(* Logix 5000 project; controller cal1632 1756-L62 rev 16.20; software revision 16.05; part 10 of 57 *)
(* tags used below, declared in another part *)
   FAULT : BOOL;
   HMI : BOOL;
   p01_sys_scp : SYS_SCP;
   p01r02 : routine;
   p01r09_pb_global_reset : BOOL;
   p11_ai_exh_amps : REAL;
   p11_ai_exh_hz : REAL;
   p11_ai_exh_hz_max : REAL;
   p11_ai_exh_rpm : REAL;
   p11_ai_lfl : REAL;
   p11_ai_prs : REAL;
   p11_ai_recirc_amps : REAL;
   p11_ai_recirc_hz : REAL;
   p11_ai_recirc_hz_max : REAL;
   p11_ai_recirc_rpm : REAL;
   p11_ai_tc01 : REAL;
   p11_ai_tc02 : REAL;
   p11_ao_cv : REAL;
   p11_ao_exhaust_selected_speed : REAL;
   p11_ao_recirc_selected_speed : REAL;
   p11_di_burner_auto : BOOL;
   p11_di_burner_safeties_ok : BOOL;
   p11_di_door_open : BOOL;
   p11_di_exh : acs800_di_normal;
   p11_di_exh_fan_mtr_ts : BOOL;
   p11_di_exh_flow_ok : BOOL;
   p11_di_flame_failure : BOOL;
   p11_di_flame_on : BOOL;
   p11_di_fresh_air_clean : BOOL;
   p11_di_high_limit_temp_ok : BOOL;
   p11_di_recirc : acs800_di_normal;
   p11_di_recirc_fan_mtr_ts : BOOL;
   p11_di_recirc_flow_ok : BOOL;
   p11_di_sp0 : BOOL;
   p11_di_sp00 : BOOL;
   p11_di_sp1 : BOOL;
   p11_di_sp2 : BOOL;
   p11_di_sp3 : BOOL;
   p11_di_tc01_bo : BOOL;
   p11_di_tc02_bo : BOOL;
   p11_di_zone_air_clean : BOOL;
   p11_dint_to_hmi : DINT[16];
   p11_do_enable_burner : BOOL;
   p11_do_exh : acs800_do_normal;
   p11_do_recirc : acs800_do_normal;
   p11_do_rst_flame : BOOL;
   p11_exhaust_input_max : REAL;
   p11_exhaust_input_min : REAL;
   p11_exhaust_output_max : REAL;
   p11_exhaust_output_min : REAL;
   p11_hc_input_max : REAL;
   p11_hc_input_min : REAL;
   p11_hc_output_max : REAL;
   p11_hc_output_min : REAL;
   p11_lfl_input_max : REAL;
   p11_lfl_input_min : REAL;
   p11_lfl_output_max : REAL;
   p11_lfl_output_min : REAL;
   p11_param_tc01z : REAL;
   p11_param_tc02z : REAL;
   p11_prs_input_max : REAL;
   p11_prs_input_min : REAL;
   p11_prs_output_max : REAL;
   p11_prs_output_min : REAL;
   p11_recirc_input_max : REAL;
   p11_recirc_input_min : REAL;
   p11_recirc_output_max : REAL;
   p11_recirc_output_min : REAL;
   p11r03 : routine;
   p11r03_hz : SYS_SCP;
   p11r03_timer_fault : TIMER[4];
   p11r03_timer_warning : TIMER[4];
   p11r04 : routine;
   p11r04_timer_fault : TIMER[4];
   p11r04_timer_warning : TIMER[4];
   p11r05 : routine;
   p11r05_exh_status : DINT;
   p11r05_recirc_status : DINT;
   p11r05_temp_ctrl_status : DINT;
   p11r05_timer_fault : TIMER[4];
   p11r05_timer_warning : TIMER[4];
   p11r20_state : DINT;
   p11r20_status : DINT;
   p11r30 : routine;
   p11r30_permissive_run : BOOL;
   p11r30_request_heat : BOOL;
   p11r30_request_manual : BOOL;
   p11r30_vfds_ready : BOOL;
   p11r31 : routine;
   p11r31_request_auto_run : BOOL;
   p11r31_request_auto_stop : BOOL;
   p11r31_vfd_stopped : BOOL;
   p11r32 : routine;
   p11r32_request_auto_run : BOOL;
   p11r32_request_auto_stop : BOOL;
   p11r32_vfd_stopped : BOOL;
(* P11_Zone_1, continued *)

ROUTINE R03_Input   (* ladder *)
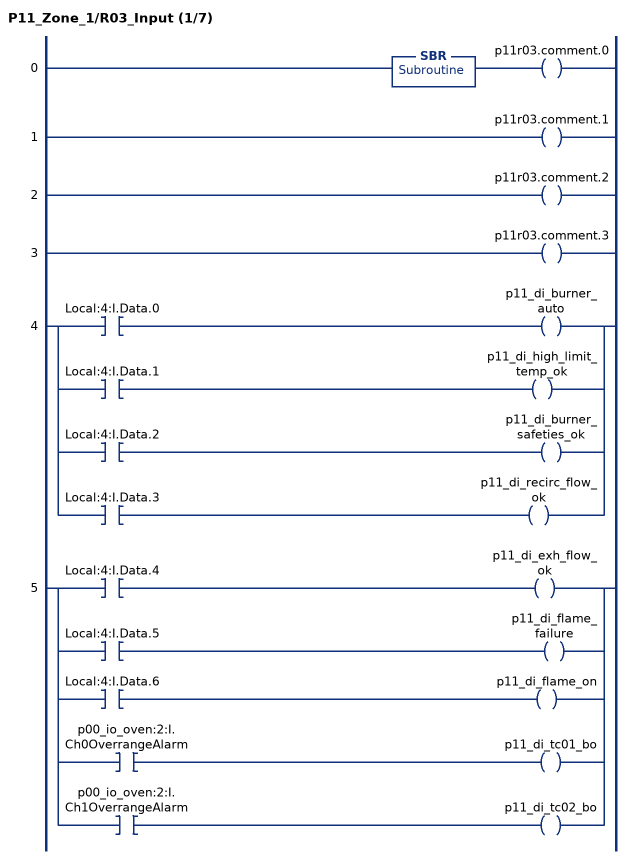
   0: SBR()OTE(p11r03.comment.0);
   1: OTE(p11r03.comment.1);
   2: OTE(p11r03.comment.2);
   3: OTE(p11r03.comment.3);
   4: [XIC(Local:4:I.Data.0) OTE(p11_di_burner_auto) ,XIC(Local:4:I.Data.1) OTE(p11_di_high_limit_temp_ok) ,XIC(Local:4:I.Data.2) OTE(p11_di_burner_safeties_ok) ,XIC(Local:4:I.Data.3) OTE(p11_di_recirc_flow_ok) ];
   5: [XIC(Local:4:I.Data.4) OTE(p11_di_exh_flow_ok) ,XIC(Local:4:I.Data.5) OTE(p11_di_flame_failure) ,XIC(Local:4:I.Data.6) OTE(p11_di_flame_on) ,XIC(p00_io_oven:2:I.Ch0OverrangeAlarm) OTE(p11_di_tc01_bo) ,XIC(p00_io_oven:2:I.Ch1OverrangeAlarm) OTE(p11_di_tc02_bo) ];
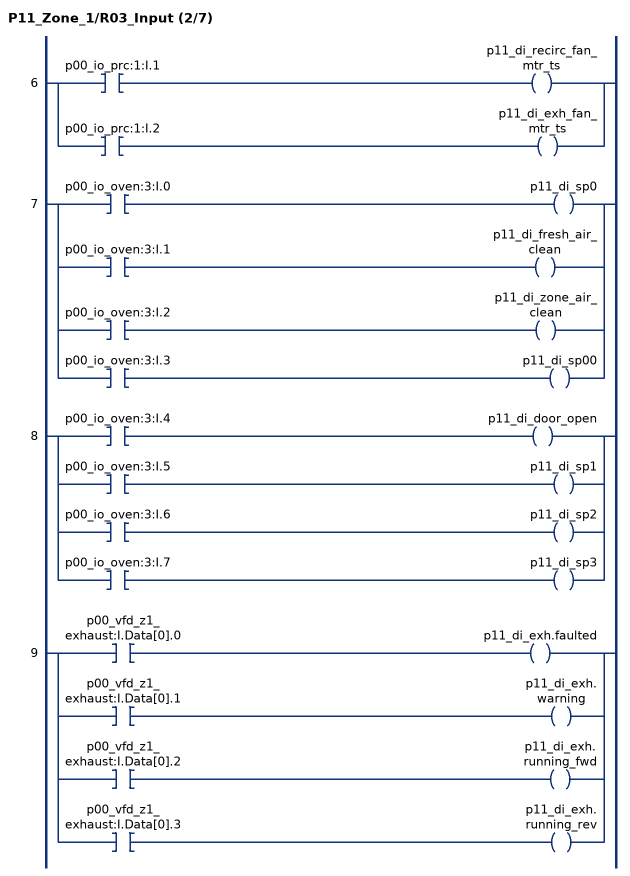
   6: [XIC(p00_io_prc:1:I.1) OTE(p11_di_recirc_fan_mtr_ts) ,XIC(p00_io_prc:1:I.2) OTE(p11_di_exh_fan_mtr_ts) ];
   7: [XIC(p00_io_oven:3:I.0) OTE(p11_di_sp0) ,XIC(p00_io_oven:3:I.1) OTE(p11_di_fresh_air_clean) ,XIC(p00_io_oven:3:I.2) OTE(p11_di_zone_air_clean) ,XIC(p00_io_oven:3:I.3) OTE(p11_di_sp00) ];
   8: [XIC(p00_io_oven:3:I.4) OTE(p11_di_door_open) ,XIC(p00_io_oven:3:I.5) OTE(p11_di_sp1) ,XIC(p00_io_oven:3:I.6) OTE(p11_di_sp2) ,XIC(p00_io_oven:3:I.7) OTE(p11_di_sp3) ];
   9: [XIC(p00_vfd_z1_exhaust:I.Data[0].0) OTE(p11_di_exh.faulted) ,XIC(p00_vfd_z1_exhaust:I.Data[0].1) OTE(p11_di_exh.warning) ,XIC(p00_vfd_z1_exhaust:I.Data[0].2) OTE(p11_di_exh.running_fwd) ,XIC(p00_vfd_z1_exhaust:I.Data[0].3) OTE(p11_di_exh.running_rev) ];
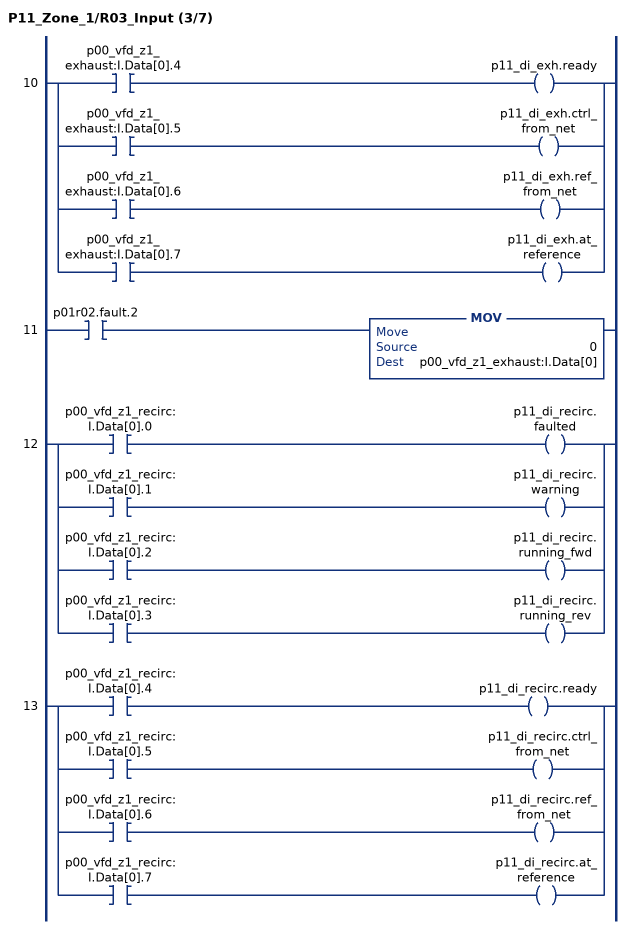
   10: [XIC(p00_vfd_z1_exhaust:I.Data[0].4) OTE(p11_di_exh.ready) ,XIC(p00_vfd_z1_exhaust:I.Data[0].5) OTE(p11_di_exh.ctrl_from_net) ,XIC(p00_vfd_z1_exhaust:I.Data[0].6) OTE(p11_di_exh.ref_from_net) ,XIC(p00_vfd_z1_exhaust:I.Data[0].7) OTE(p11_di_exh.at_reference) ];
   11: XIC(p01r02.fault.2)MOV(0,p00_vfd_z1_exhaust:I.Data[0]);
   12: [XIC(p00_vfd_z1_recirc:I.Data[0].0) OTE(p11_di_recirc.faulted) ,XIC(p00_vfd_z1_recirc:I.Data[0].1) OTE(p11_di_recirc.warning) ,XIC(p00_vfd_z1_recirc:I.Data[0].2) OTE(p11_di_recirc.running_fwd) ,XIC(p00_vfd_z1_recirc:I.Data[0].3) OTE(p11_di_recirc.running_rev) ];
   13: [XIC(p00_vfd_z1_recirc:I.Data[0].4) OTE(p11_di_recirc.ready) ,XIC(p00_vfd_z1_recirc:I.Data[0].5) OTE(p11_di_recirc.ctrl_from_net) ,XIC(p00_vfd_z1_recirc:I.Data[0].6) OTE(p11_di_recirc.ref_from_net) ,XIC(p00_vfd_z1_recirc:I.Data[0].7) OTE(p11_di_recirc.at_reference) ];
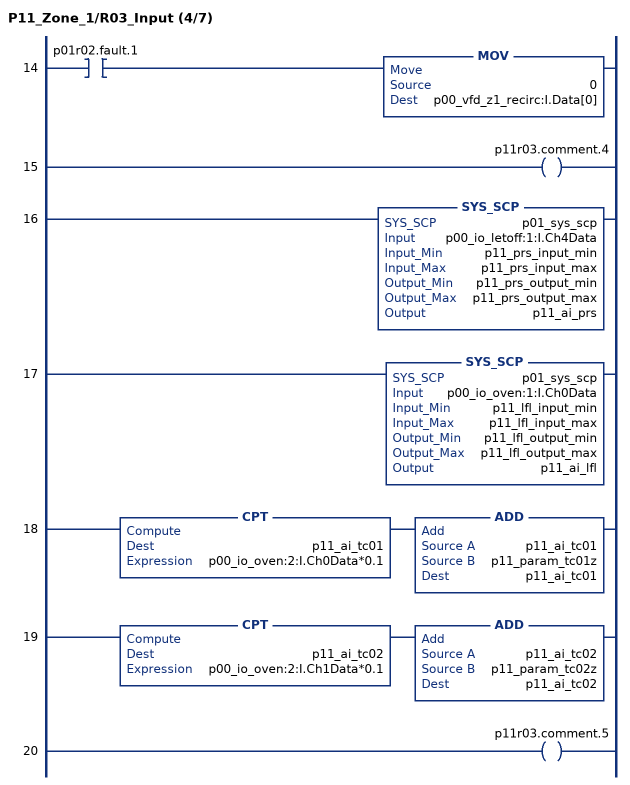
   14: XIC(p01r02.fault.1)MOV(0,p00_vfd_z1_recirc:I.Data[0]);
   15: OTE(p11r03.comment.4);
   16: SYS_SCP(p01_sys_scp,p00_io_letoff:1:I.Ch4Data,p11_prs_input_min,p11_prs_input_max,p11_prs_output_min,p11_prs_output_max,p11_ai_prs);
   17: SYS_SCP(p01_sys_scp,p00_io_oven:1:I.Ch0Data,p11_lfl_input_min,p11_lfl_input_max,p11_lfl_output_min,p11_lfl_output_max,p11_ai_lfl);
   18: CPT(p11_ai_tc01,p00_io_oven:2:I.Ch0Data*0.1)ADD(p11_ai_tc01,p11_param_tc01z,p11_ai_tc01);
   19: CPT(p11_ai_tc02,p00_io_oven:2:I.Ch1Data*0.1)ADD(p11_ai_tc02,p11_param_tc02z,p11_ai_tc02);
   20: OTE(p11r03.comment.5);
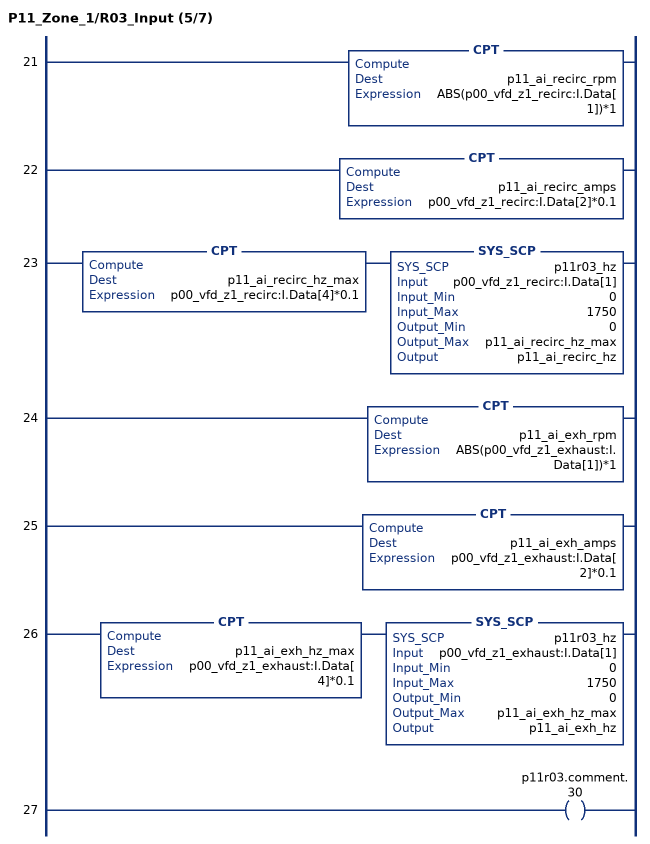
   21: CPT(p11_ai_recirc_rpm,ABS(p00_vfd_z1_recirc:I.Data[1])*1);
   22: CPT(p11_ai_recirc_amps,p00_vfd_z1_recirc:I.Data[2]*0.1);
   23: CPT(p11_ai_recirc_hz_max,p00_vfd_z1_recirc:I.Data[4]*0.1)SYS_SCP(p11r03_hz,p00_vfd_z1_recirc:I.Data[1],0,1750,0,p11_ai_recirc_hz_max,p11_ai_recirc_hz);
   24: CPT(p11_ai_exh_rpm,ABS(p00_vfd_z1_exhaust:I.Data[1])*1);
   25: CPT(p11_ai_exh_amps,p00_vfd_z1_exhaust:I.Data[2]*0.1);
   26: CPT(p11_ai_exh_hz_max,p00_vfd_z1_exhaust:I.Data[4]*0.1)SYS_SCP(p11r03_hz,p00_vfd_z1_exhaust:I.Data[1],0,1750,0,p11_ai_exh_hz_max,p11_ai_exh_hz);
   27: OTE(p11r03.comment.30);
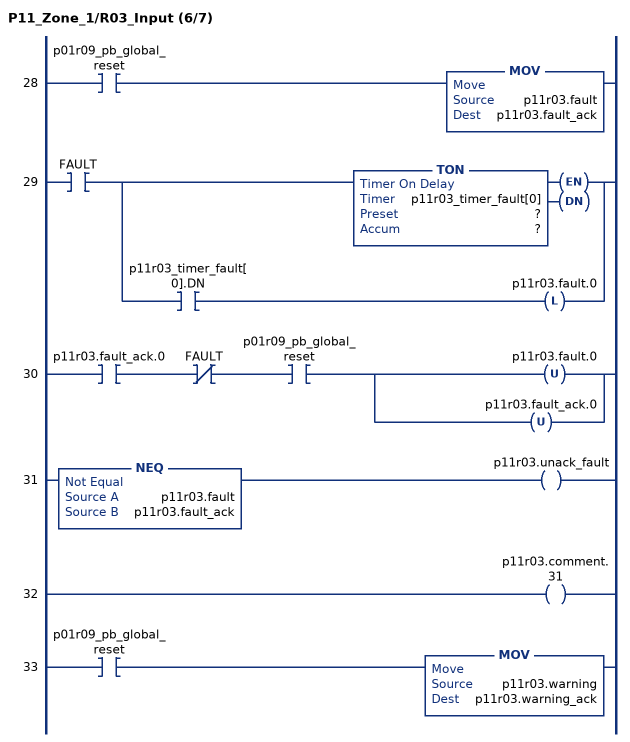
   28: XIC(p01r09_pb_global_reset)MOV(p11r03.fault,p11r03.fault_ack);
   29: XIC(FAULT)[TON(p11r03_timer_fault[0],?,?) ,XIC(p11r03_timer_fault[0].DN) OTL(p11r03.fault.0) ];
   30: XIC(p11r03.fault_ack.0)XIO(FAULT)XIC(p01r09_pb_global_reset)[OTU(p11r03.fault.0) ,OTU(p11r03.fault_ack.0) ];
   31: NEQ(p11r03.fault,p11r03.fault_ack)OTE(p11r03.unack_fault);
   32: OTE(p11r03.comment.31);
   33: XIC(p01r09_pb_global_reset)MOV(p11r03.warning,p11r03.warning_ack);
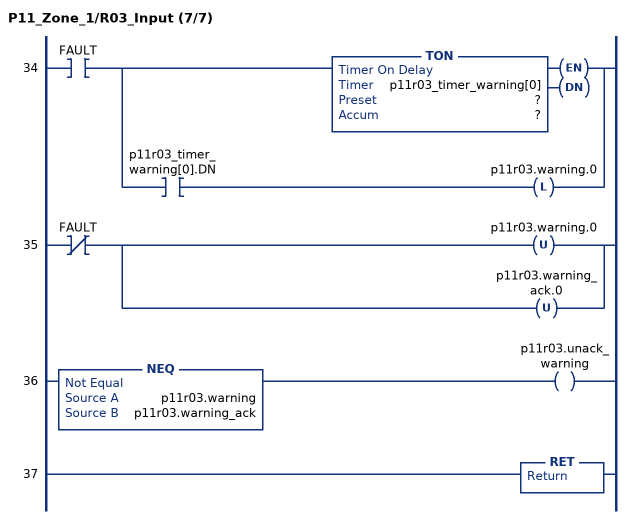
   34: XIC(FAULT)[TON(p11r03_timer_warning[0],?,?) ,XIC(p11r03_timer_warning[0].DN) OTL(p11r03.warning.0) ];
   35: XIO(FAULT)[OTU(p11r03.warning.0) ,OTU(p11r03.warning_ack.0) ];
   36: NEQ(p11r03.warning,p11r03.warning_ack)OTE(p11r03.unack_warning);
   37: RET();
END_ROUTINE

ROUTINE R04_Output   (* ladder *)
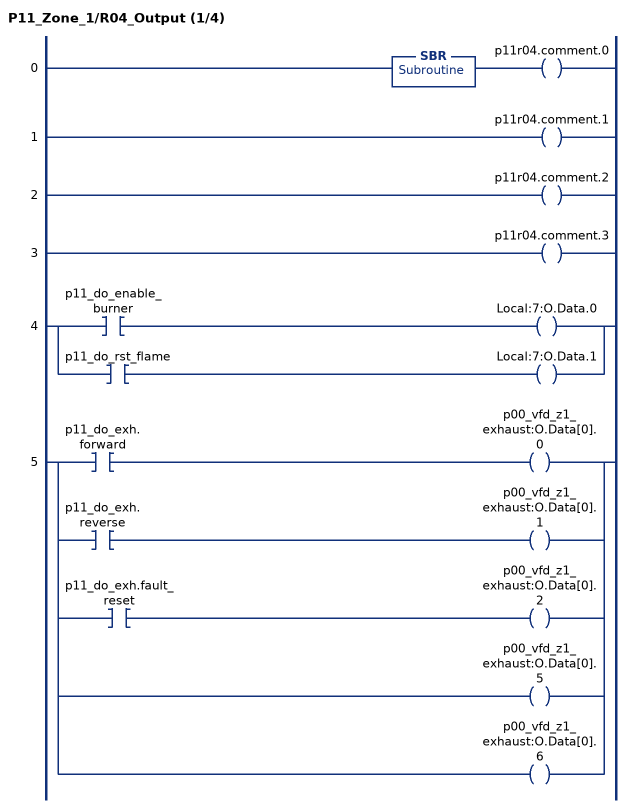
   0: SBR()OTE(p11r04.comment.0);
   1: OTE(p11r04.comment.1);
   2: OTE(p11r04.comment.2);
   3: OTE(p11r04.comment.3);
   4: [XIC(p11_do_enable_burner) OTE(Local:7:O.Data.0) ,XIC(p11_do_rst_flame) OTE(Local:7:O.Data.1) ];
   5: [XIC(p11_do_exh.forward) OTE(p00_vfd_z1_exhaust:O.Data[0].0) ,XIC(p11_do_exh.reverse) OTE(p00_vfd_z1_exhaust:O.Data[0].1) ,XIC(p11_do_exh.fault_reset) OTE(p00_vfd_z1_exhaust:O.Data[0].2) ,OTE(p00_vfd_z1_exhaust:O.Data[0].5) ,OTE(p00_vfd_z1_exhaust:O.Data[0].6) ];
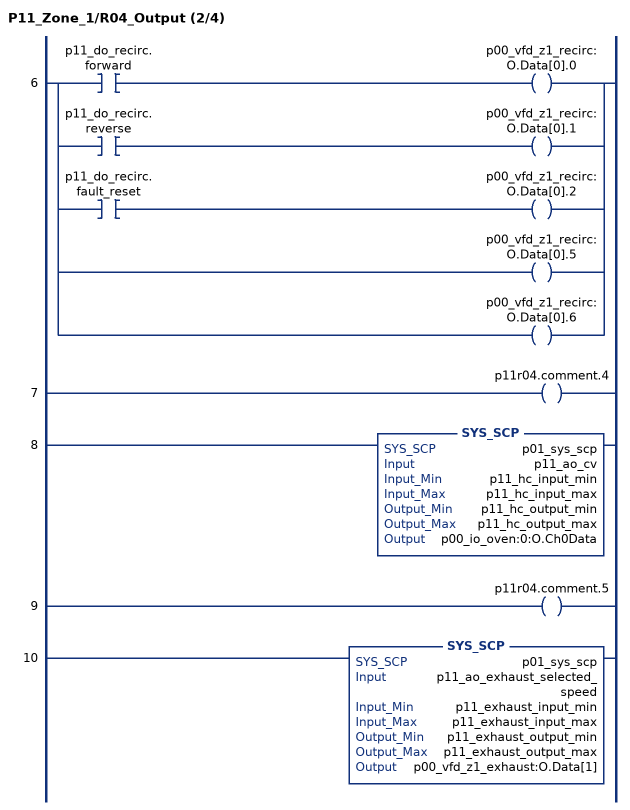
   6: [XIC(p11_do_recirc.forward) OTE(p00_vfd_z1_recirc:O.Data[0].0) ,XIC(p11_do_recirc.reverse) OTE(p00_vfd_z1_recirc:O.Data[0].1) ,XIC(p11_do_recirc.fault_reset) OTE(p00_vfd_z1_recirc:O.Data[0].2) ,OTE(p00_vfd_z1_recirc:O.Data[0].5) ,OTE(p00_vfd_z1_recirc:O.Data[0].6) ];
   7: OTE(p11r04.comment.4);
   8: SYS_SCP(p01_sys_scp,p11_ao_cv,p11_hc_input_min,p11_hc_input_max,p11_hc_output_min,p11_hc_output_max,p00_io_oven:0:O.Ch0Data);
   9: OTE(p11r04.comment.5);
   10: SYS_SCP(p01_sys_scp,p11_ao_exhaust_selected_speed,p11_exhaust_input_min,p11_exhaust_input_max,p11_exhaust_output_min,p11_exhaust_output_max,p00_vfd_z1_exhaust:O.Data[1]);
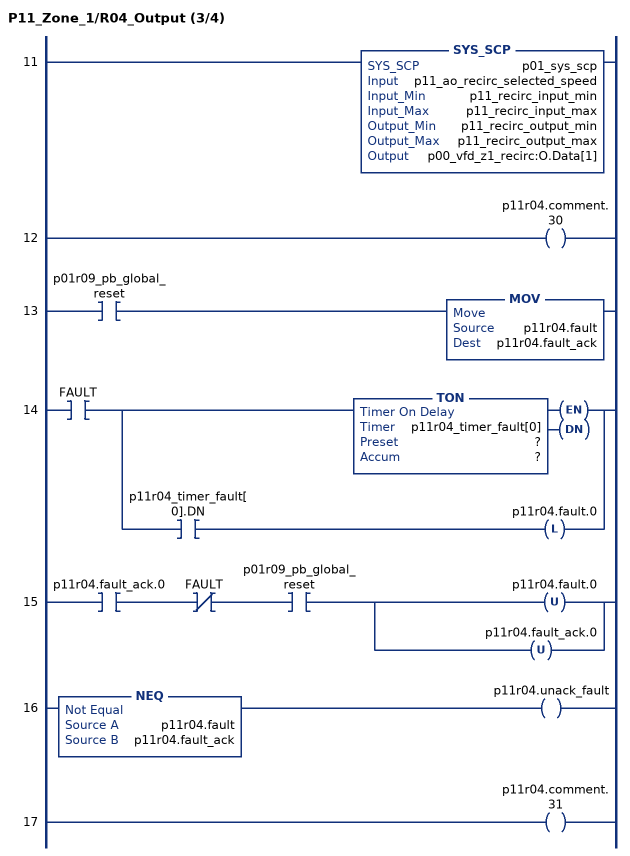
   11: SYS_SCP(p01_sys_scp,p11_ao_recirc_selected_speed,p11_recirc_input_min,p11_recirc_input_max,p11_recirc_output_min,p11_recirc_output_max,p00_vfd_z1_recirc:O.Data[1]);
   12: OTE(p11r04.comment.30);
   13: XIC(p01r09_pb_global_reset)MOV(p11r04.fault,p11r04.fault_ack);
   14: XIC(FAULT)[TON(p11r04_timer_fault[0],?,?) ,XIC(p11r04_timer_fault[0].DN) OTL(p11r04.fault.0) ];
   15: XIC(p11r04.fault_ack.0)XIO(FAULT)XIC(p01r09_pb_global_reset)[OTU(p11r04.fault.0) ,OTU(p11r04.fault_ack.0) ];
   16: NEQ(p11r04.fault,p11r04.fault_ack)OTE(p11r04.unack_fault);
   17: OTE(p11r04.comment.31);
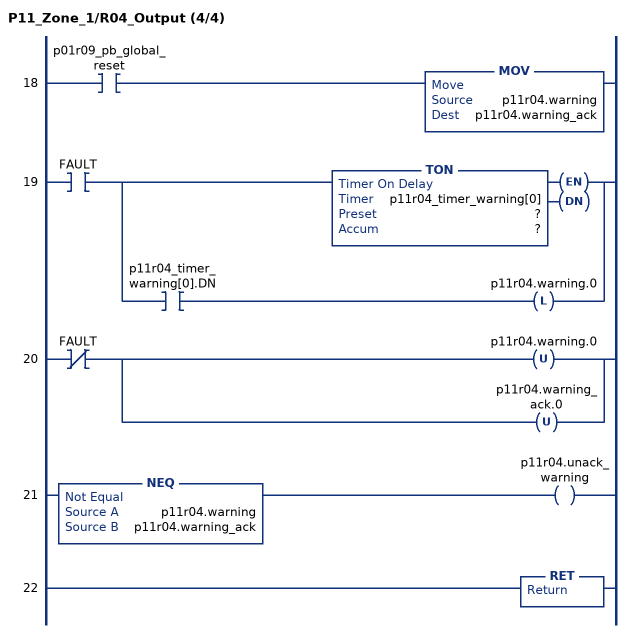
   18: XIC(p01r09_pb_global_reset)MOV(p11r04.warning,p11r04.warning_ack);
   19: XIC(FAULT)[TON(p11r04_timer_warning[0],?,?) ,XIC(p11r04_timer_warning[0].DN) OTL(p11r04.warning.0) ];
   20: XIO(FAULT)[OTU(p11r04.warning.0) ,OTU(p11r04.warning_ack.0) ];
   21: NEQ(p11r04.warning,p11r04.warning_ack)OTE(p11r04.unack_warning);
   22: RET();
END_ROUTINE

ROUTINE R05_Dint_to_HMI   (* ladder *)
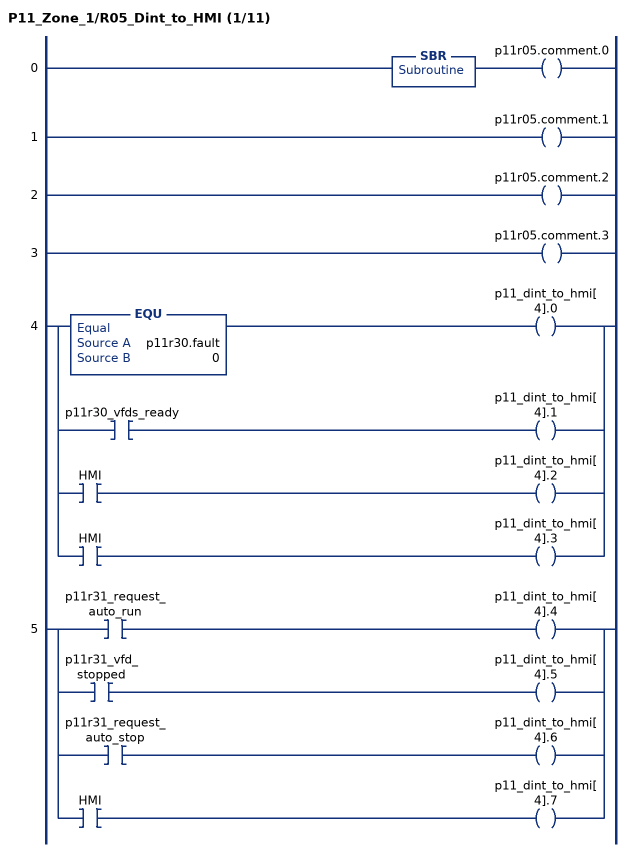
   0: SBR()OTE(p11r05.comment.0);
   1: OTE(p11r05.comment.1);
   2: OTE(p11r05.comment.2);
   3: OTE(p11r05.comment.3);
   4: [EQU(p11r30.fault,0) OTE(p11_dint_to_hmi[4].0) ,XIC(p11r30_vfds_ready) OTE(p11_dint_to_hmi[4].1) ,XIC(HMI) OTE(p11_dint_to_hmi[4].2) ,XIC(HMI) OTE(p11_dint_to_hmi[4].3) ];
   5: [XIC(p11r31_request_auto_run) OTE(p11_dint_to_hmi[4].4) ,XIC(p11r31_vfd_stopped) OTE(p11_dint_to_hmi[4].5) ,XIC(p11r31_request_auto_stop) OTE(p11_dint_to_hmi[4].6) ,XIC(HMI) OTE(p11_dint_to_hmi[4].7) ];
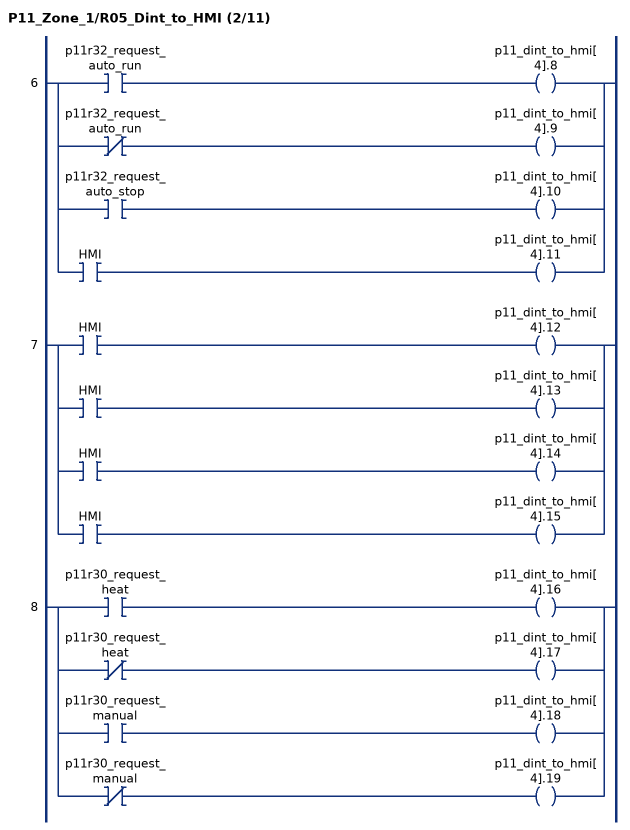
   6: [XIC(p11r32_request_auto_run) OTE(p11_dint_to_hmi[4].8) ,XIO(p11r32_request_auto_run) OTE(p11_dint_to_hmi[4].9) ,XIC(p11r32_request_auto_stop) OTE(p11_dint_to_hmi[4].10) ,XIC(HMI) OTE(p11_dint_to_hmi[4].11) ];
   7: [XIC(HMI) OTE(p11_dint_to_hmi[4].12) ,XIC(HMI) OTE(p11_dint_to_hmi[4].13) ,XIC(HMI) OTE(p11_dint_to_hmi[4].14) ,XIC(HMI) OTE(p11_dint_to_hmi[4].15) ];
   8: [XIC(p11r30_request_heat) OTE(p11_dint_to_hmi[4].16) ,XIO(p11r30_request_heat) OTE(p11_dint_to_hmi[4].17) ,XIC(p11r30_request_manual) OTE(p11_dint_to_hmi[4].18) ,XIO(p11r30_request_manual) OTE(p11_dint_to_hmi[4].19) ];
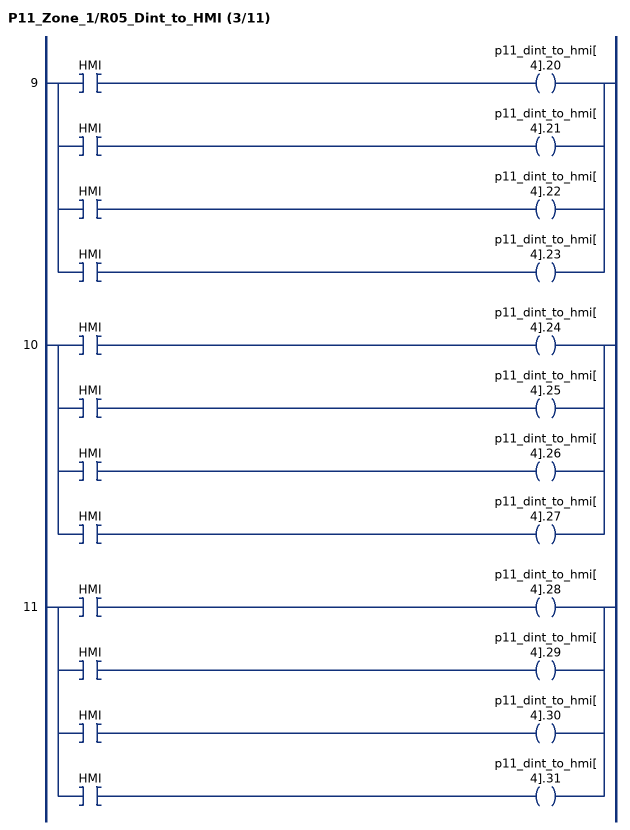
   9: [XIC(HMI) OTE(p11_dint_to_hmi[4].20) ,XIC(HMI) OTE(p11_dint_to_hmi[4].21) ,XIC(HMI) OTE(p11_dint_to_hmi[4].22) ,XIC(HMI) OTE(p11_dint_to_hmi[4].23) ];
   10: [XIC(HMI) OTE(p11_dint_to_hmi[4].24) ,XIC(HMI) OTE(p11_dint_to_hmi[4].25) ,XIC(HMI) OTE(p11_dint_to_hmi[4].26) ,XIC(HMI) OTE(p11_dint_to_hmi[4].27) ];
   11: [XIC(HMI) OTE(p11_dint_to_hmi[4].28) ,XIC(HMI) OTE(p11_dint_to_hmi[4].29) ,XIC(HMI) OTE(p11_dint_to_hmi[4].30) ,XIC(HMI) OTE(p11_dint_to_hmi[4].31) ];
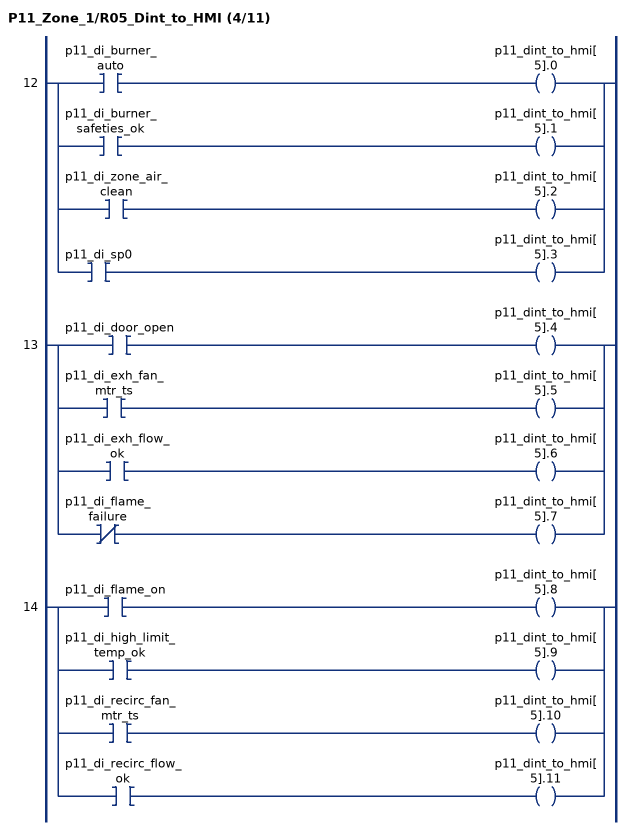
   12: [XIC(p11_di_burner_auto) OTE(p11_dint_to_hmi[5].0) ,XIC(p11_di_burner_safeties_ok) OTE(p11_dint_to_hmi[5].1) ,XIC(p11_di_zone_air_clean) OTE(p11_dint_to_hmi[5].2) ,XIC(p11_di_sp0) OTE(p11_dint_to_hmi[5].3) ];
   13: [XIC(p11_di_door_open) OTE(p11_dint_to_hmi[5].4) ,XIC(p11_di_exh_fan_mtr_ts) OTE(p11_dint_to_hmi[5].5) ,XIC(p11_di_exh_flow_ok) OTE(p11_dint_to_hmi[5].6) ,XIO(p11_di_flame_failure) OTE(p11_dint_to_hmi[5].7) ];
   14: [XIC(p11_di_flame_on) OTE(p11_dint_to_hmi[5].8) ,XIC(p11_di_high_limit_temp_ok) OTE(p11_dint_to_hmi[5].9) ,XIC(p11_di_recirc_fan_mtr_ts) OTE(p11_dint_to_hmi[5].10) ,XIC(p11_di_recirc_flow_ok) OTE(p11_dint_to_hmi[5].11) ];
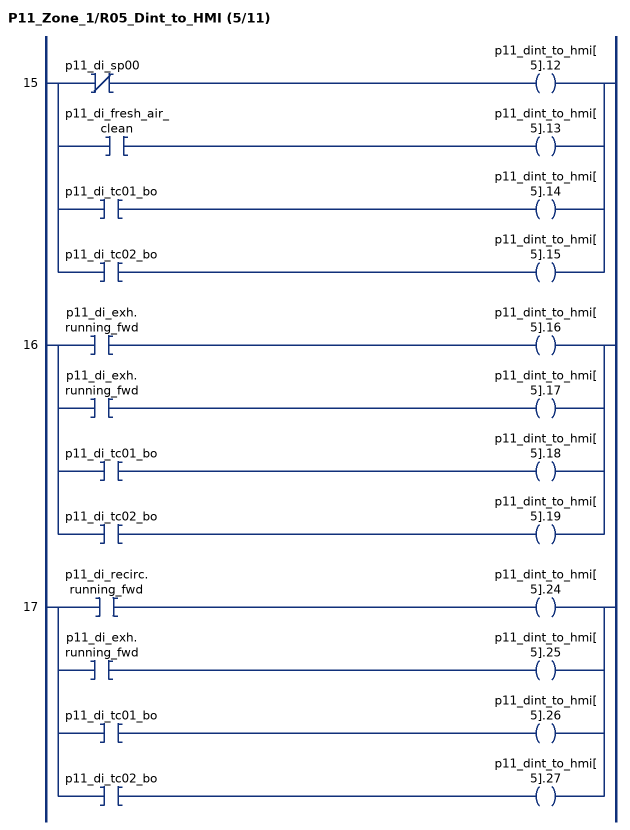
   15: [XIO(p11_di_sp00) OTE(p11_dint_to_hmi[5].12) ,XIC(p11_di_fresh_air_clean) OTE(p11_dint_to_hmi[5].13) ,XIC(p11_di_tc01_bo) OTE(p11_dint_to_hmi[5].14) ,XIC(p11_di_tc02_bo) OTE(p11_dint_to_hmi[5].15) ];
   16: [XIC(p11_di_exh.running_fwd) OTE(p11_dint_to_hmi[5].16) ,XIC(p11_di_exh.running_fwd) OTE(p11_dint_to_hmi[5].17) ,XIC(p11_di_tc01_bo) OTE(p11_dint_to_hmi[5].18) ,XIC(p11_di_tc02_bo) OTE(p11_dint_to_hmi[5].19) ];
   17: [XIC(p11_di_recirc.running_fwd) OTE(p11_dint_to_hmi[5].24) ,XIC(p11_di_exh.running_fwd) OTE(p11_dint_to_hmi[5].25) ,XIC(p11_di_tc01_bo) OTE(p11_dint_to_hmi[5].26) ,XIC(p11_di_tc02_bo) OTE(p11_dint_to_hmi[5].27) ];
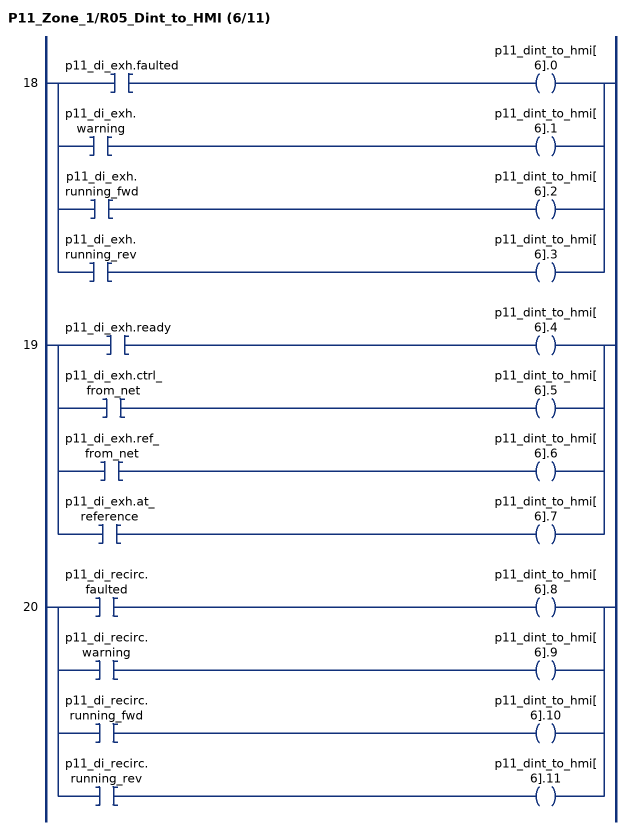
   18: [XIC(p11_di_exh.faulted) OTE(p11_dint_to_hmi[6].0) ,XIC(p11_di_exh.warning) OTE(p11_dint_to_hmi[6].1) ,XIC(p11_di_exh.running_fwd) OTE(p11_dint_to_hmi[6].2) ,XIC(p11_di_exh.running_rev) OTE(p11_dint_to_hmi[6].3) ];
   19: [XIC(p11_di_exh.ready) OTE(p11_dint_to_hmi[6].4) ,XIC(p11_di_exh.ctrl_from_net) OTE(p11_dint_to_hmi[6].5) ,XIC(p11_di_exh.ref_from_net) OTE(p11_dint_to_hmi[6].6) ,XIC(p11_di_exh.at_reference) OTE(p11_dint_to_hmi[6].7) ];
   20: [XIC(p11_di_recirc.faulted) OTE(p11_dint_to_hmi[6].8) ,XIC(p11_di_recirc.warning) OTE(p11_dint_to_hmi[6].9) ,XIC(p11_di_recirc.running_fwd) OTE(p11_dint_to_hmi[6].10) ,XIC(p11_di_recirc.running_rev) OTE(p11_dint_to_hmi[6].11) ];
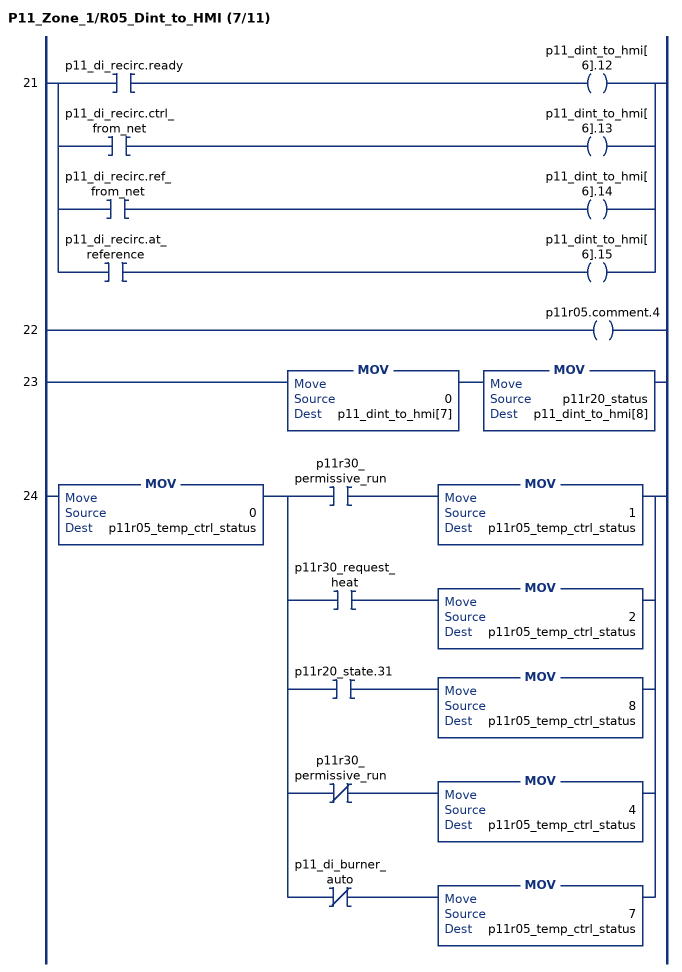
   21: [XIC(p11_di_recirc.ready) OTE(p11_dint_to_hmi[6].12) ,XIC(p11_di_recirc.ctrl_from_net) OTE(p11_dint_to_hmi[6].13) ,XIC(p11_di_recirc.ref_from_net) OTE(p11_dint_to_hmi[6].14) ,XIC(p11_di_recirc.at_reference) OTE(p11_dint_to_hmi[6].15) ];
   22: OTE(p11r05.comment.4);
   23: MOV(0,p11_dint_to_hmi[7])MOV(p11r20_status,p11_dint_to_hmi[8]);
   24: MOV(0,p11r05_temp_ctrl_status)[XIC(p11r30_permissive_run) MOV(1,p11r05_temp_ctrl_status) ,XIC(p11r30_request_heat) MOV(2,p11r05_temp_ctrl_status) ,XIC(p11r20_state.31) MOV(8,p11r05_temp_ctrl_status) ,XIO(p11r30_permissive_run) MOV(4,p11r05_temp_ctrl_status) ,XIO(p11_di_burner_auto) MOV(7,p11r05_temp_ctrl_status) ];
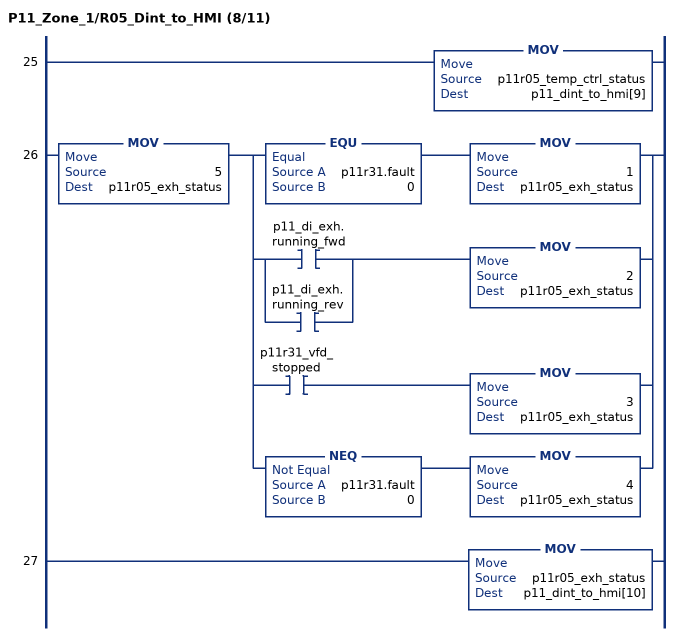
   25: MOV(p11r05_temp_ctrl_status,p11_dint_to_hmi[9]);
   26: MOV(5,p11r05_exh_status)[EQU(p11r31.fault,0) MOV(1,p11r05_exh_status) ,[XIC(p11_di_exh.running_fwd) ,XIC(p11_di_exh.running_rev) ] MOV(2,p11r05_exh_status) ,XIC(p11r31_vfd_stopped) MOV(3,p11r05_exh_status) ,NEQ(p11r31.fault,0) MOV(4,p11r05_exh_status) ];
   27: MOV(p11r05_exh_status,p11_dint_to_hmi[10]);
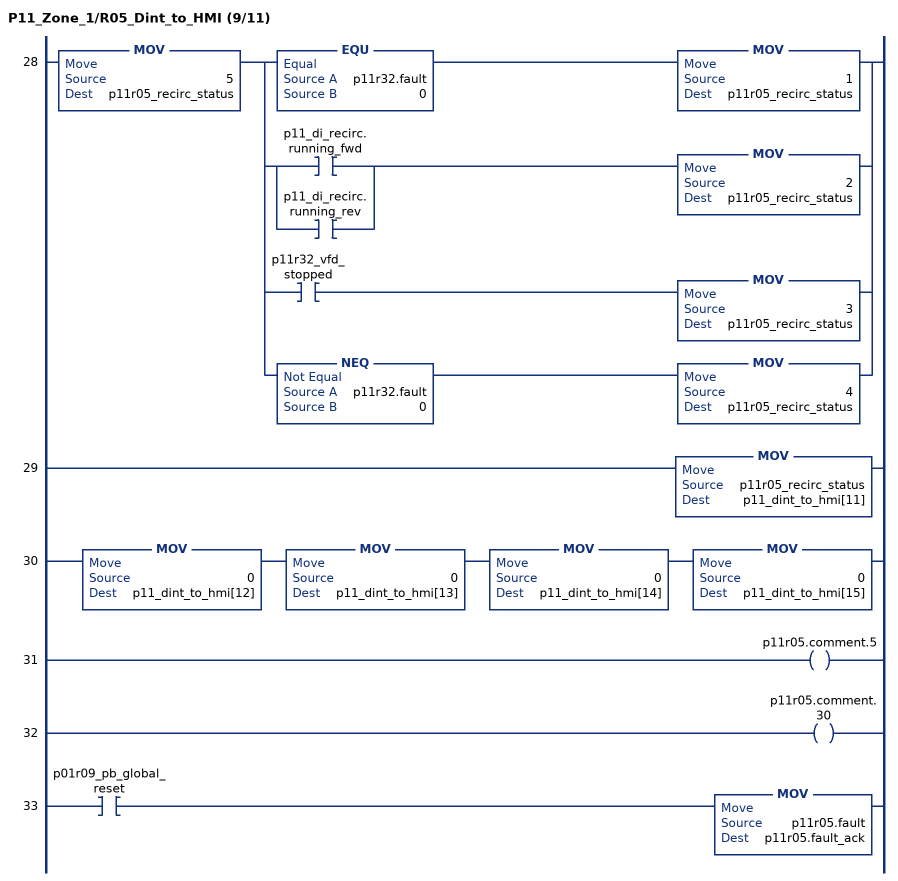
   28: MOV(5,p11r05_recirc_status)[EQU(p11r32.fault,0) MOV(1,p11r05_recirc_status) ,[XIC(p11_di_recirc.running_fwd) ,XIC(p11_di_recirc.running_rev) ] MOV(2,p11r05_recirc_status) ,XIC(p11r32_vfd_stopped) MOV(3,p11r05_recirc_status) ,NEQ(p11r32.fault,0) MOV(4,p11r05_recirc_status) ];
   29: MOV(p11r05_recirc_status,p11_dint_to_hmi[11]);
   30: MOV(0,p11_dint_to_hmi[12])MOV(0,p11_dint_to_hmi[13])MOV(0,p11_dint_to_hmi[14])MOV(0,p11_dint_to_hmi[15]);
   31: OTE(p11r05.comment.5);
   32: OTE(p11r05.comment.30);
   33: XIC(p01r09_pb_global_reset)MOV(p11r05.fault,p11r05.fault_ack);
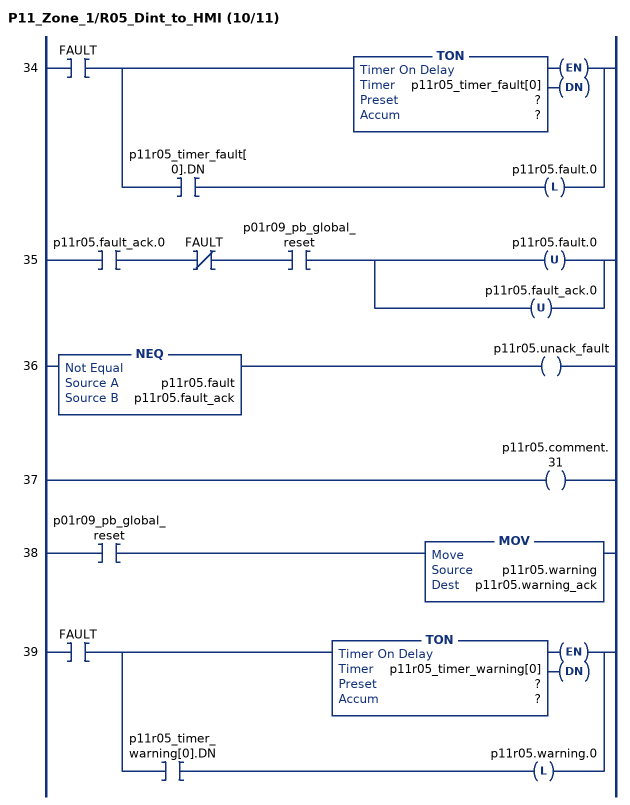
   34: XIC(FAULT)[TON(p11r05_timer_fault[0],?,?) ,XIC(p11r05_timer_fault[0].DN) OTL(p11r05.fault.0) ];
   35: XIC(p11r05.fault_ack.0)XIO(FAULT)XIC(p01r09_pb_global_reset)[OTU(p11r05.fault.0) ,OTU(p11r05.fault_ack.0) ];
   36: NEQ(p11r05.fault,p11r05.fault_ack)OTE(p11r05.unack_fault);
   37: OTE(p11r05.comment.31);
   38: XIC(p01r09_pb_global_reset)MOV(p11r05.warning,p11r05.warning_ack);
   39: XIC(FAULT)[TON(p11r05_timer_warning[0],?,?) ,XIC(p11r05_timer_warning[0].DN) OTL(p11r05.warning.0) ];
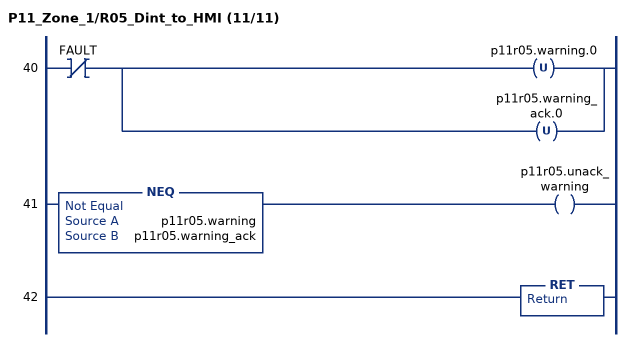
   40: XIO(FAULT)[OTU(p11r05.warning.0) ,OTU(p11r05.warning_ack.0) ];
   41: NEQ(p11r05.warning,p11r05.warning_ack)OTE(p11r05.unack_warning);
   42: RET();
END_ROUTINE
